# EPICS substitutions: epics/db/indraDrive.substitutions
file "./db/ecSlave.template"
{
  pattern {}
          {}
}

# No custom data yet
#file "./db/indraDrive.template"
#{
#  pattern {}
#          {}
#}
